REGION Network 47: Ejectors selection
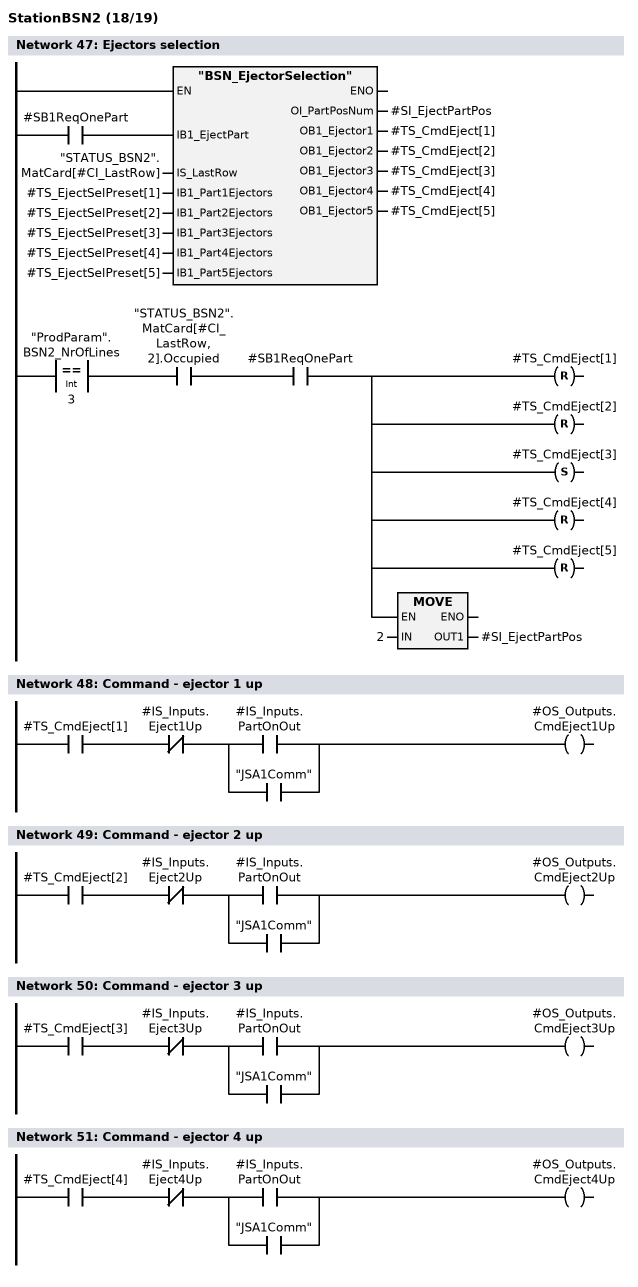
   RUNG wire#powerrail
      "BSN_EjectorSelection"(IB1_EjectPart := wire#w1, IS_LastRow := "STATUS_BSN2".MatCard[#CI_LastRow], IB1_Part1Ejectors := #TS_EjectSelPreset[1], IB1_Part2Ejectors := #TS_EjectSelPreset[2], IB1_Part3Ejectors := #TS_EjectSelPreset[3], IB1_Part4Ejectors := #TS_EjectSelPreset[4], IB1_Part5Ejectors := #TS_EjectSelPreset[5], OI_PartPosNum => #SI_EjectPartPos, OB1_Ejector1 => #TS_CmdEject[1], OB1_Ejector2 => #TS_CmdEject[2], OB1_Ejector3 => #TS_CmdEject[3], OB1_Ejector4 => #TS_CmdEject[4], OB1_Ejector5 => #TS_CmdEject[5])
   END_RUNG
   RUNG wire#powerrail
      Contact( #SB1ReqOnePart )
   END_RUNG wire#w1
   RUNG wire#powerrail
      { S7_Templates := "SrcType := Int" } EQ_Contact(in1 := "ProdParam".BSN2_NrOfLines, in2 := 3)
      Contact( "STATUS_BSN2".MatCard[#CI_LastRow, 2].Occupied )
      Contact( #SB1ReqOnePart )
      wire#w2
      R_Coil( #TS_CmdEject[1] )
   END_RUNG
   RUNG wire#w2
      R_Coil( #TS_CmdEject[2] )
   END_RUNG
   RUNG wire#w2
      S_Coil( #TS_CmdEject[3] )
   END_RUNG
   RUNG wire#w2
      R_Coil( #TS_CmdEject[4] )
   END_RUNG
   RUNG wire#w2
      R_Coil( #TS_CmdEject[5] )
   END_RUNG
   RUNG wire#w2
      Move(in := 2, out1 => #SI_EjectPartPos)
   END_RUNG
   // the same network as SCL:
   "BSN_EjectorSelection"(IB1_EjectPart := #SB1ReqOnePart,
                          IS_LastRow := "STATUS_BSN2".MatCard[#CI_LastRow],
                          IB1_Part1Ejectors := #TS_EjectSelPreset[1],
                          IB1_Part2Ejectors := #TS_EjectSelPreset[2],
                          IB1_Part3Ejectors := #TS_EjectSelPreset[3],
                          IB1_Part4Ejectors := #TS_EjectSelPreset[4],
                          IB1_Part5Ejectors := #TS_EjectSelPreset[5],
                          OI_PartPosNum => #SI_EjectPartPos,
                          OB1_Ejector1 => #TS_CmdEject[1],
                          OB1_Ejector2 => #TS_CmdEject[2],
                          OB1_Ejector3 => #TS_CmdEject[3],
                          OB1_Ejector4 => #TS_CmdEject[4],
                          OB1_Ejector5 => #TS_CmdEject[5]);
   IF ("ProdParam".BSN2_NrOfLines = 3) AND "STATUS_BSN2".MatCard[#CI_LastRow, 2].Occupied AND #SB1ReqOnePart THEN
       #TS_CmdEject[1] := FALSE;
       #TS_CmdEject[2] := FALSE;
       #TS_CmdEject[3] := TRUE;
       #TS_CmdEject[4] := FALSE;
       #TS_CmdEject[5] := FALSE;
       #SI_EjectPartPos := 2;
   END_IF;
END_REGION

REGION Network 48: Command - ejector 1 up
   RUNG wire#powerrail
      Contact( #TS_CmdEject[1] )
      I_Contact( #IS_Inputs.Eject1Up )
      wire#w1
      Contact( #IS_Inputs.PartOnOut )
      wire#w2
      Coil( #OS_Outputs.CmdEject1Up )
   END_RUNG
   RUNG wire#w1
      Contact( "JSA1Comm" )
   END_RUNG wire#w2
   // the same network as SCL:
   #OS_Outputs.CmdEject1Up := #TS_CmdEject[1] AND NOT #IS_Inputs.Eject1Up AND (#IS_Inputs.PartOnOut OR "JSA1Comm");
END_REGION

REGION Network 49: Command - ejector 2 up
   RUNG wire#powerrail
      Contact( #TS_CmdEject[2] )
      I_Contact( #IS_Inputs.Eject2Up )
      wire#w1
      Contact( #IS_Inputs.PartOnOut )
      wire#w2
      Coil( #OS_Outputs.CmdEject2Up )
   END_RUNG
   RUNG wire#w1
      Contact( "JSA1Comm" )
   END_RUNG wire#w2
   // the same network as SCL:
   #OS_Outputs.CmdEject2Up := #TS_CmdEject[2] AND NOT #IS_Inputs.Eject2Up AND (#IS_Inputs.PartOnOut OR "JSA1Comm");
END_REGION

REGION Network 50: Command - ejector 3 up
   RUNG wire#powerrail
      Contact( #TS_CmdEject[3] )
      I_Contact( #IS_Inputs.Eject3Up )
      wire#w1
      Contact( #IS_Inputs.PartOnOut )
      wire#w2
      Coil( #OS_Outputs.CmdEject3Up )
   END_RUNG
   RUNG wire#w1
      Contact( "JSA1Comm" )
   END_RUNG wire#w2
   // the same network as SCL:
   #OS_Outputs.CmdEject3Up := #TS_CmdEject[3] AND NOT #IS_Inputs.Eject3Up AND (#IS_Inputs.PartOnOut OR "JSA1Comm");
END_REGION

REGION Network 51: Command - ejector 4 up
   RUNG wire#powerrail
      Contact( #TS_CmdEject[4] )
      I_Contact( #IS_Inputs.Eject4Up )
      wire#w1
      Contact( #IS_Inputs.PartOnOut )
      wire#w2
      Coil( #OS_Outputs.CmdEject4Up )
   END_RUNG
   RUNG wire#w1
      Contact( "JSA1Comm" )
   END_RUNG wire#w2
   // the same network as SCL:
   #OS_Outputs.CmdEject4Up := #TS_CmdEject[4] AND NOT #IS_Inputs.Eject4Up AND (#IS_Inputs.PartOnOut OR "JSA1Comm");
END_REGION

REGION Network 52: Command - ejector 5 up
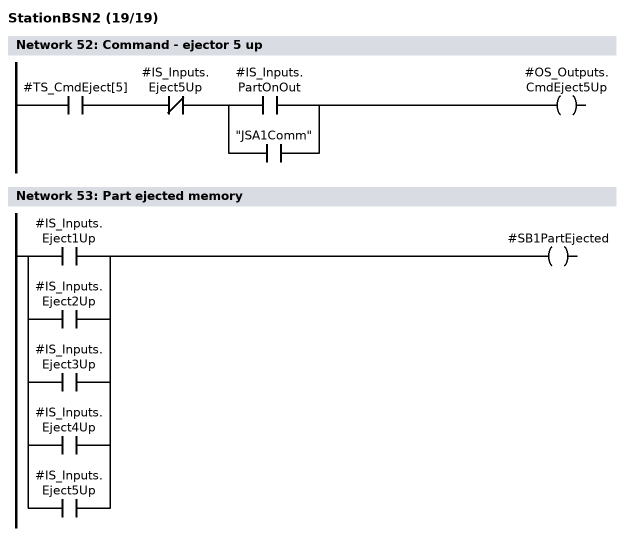
   RUNG wire#powerrail
      Contact( #TS_CmdEject[5] )
      I_Contact( #IS_Inputs.Eject5Up )
      wire#w1
      Contact( #IS_Inputs.PartOnOut )
      wire#w2
      Coil( #OS_Outputs.CmdEject5Up )
   END_RUNG
   RUNG wire#w1
      Contact( "JSA1Comm" )
   END_RUNG wire#w2
   // the same network as SCL:
   #OS_Outputs.CmdEject5Up := #TS_CmdEject[5] AND NOT #IS_Inputs.Eject5Up AND (#IS_Inputs.PartOnOut OR "JSA1Comm");
END_REGION

REGION Network 53: Part ejected memory
   RUNG wire#powerrail
      Contact( #IS_Inputs.Eject1Up )
      wire#w1
      Coil( #SB1PartEjected )
   END_RUNG
   RUNG wire#powerrail
      Contact( #IS_Inputs.Eject2Up )
   END_RUNG wire#w1
   RUNG wire#powerrail
      Contact( #IS_Inputs.Eject3Up )
   END_RUNG wire#w1
   RUNG wire#powerrail
      Contact( #IS_Inputs.Eject4Up )
   END_RUNG wire#w1
   RUNG wire#powerrail
      Contact( #IS_Inputs.Eject5Up )
   END_RUNG wire#w1
   // the same network as SCL:
   #SB1PartEjected := #IS_Inputs.Eject1Up OR #IS_Inputs.Eject2Up OR #IS_Inputs.Eject3Up OR #IS_Inputs.Eject4Up OR #IS_Inputs.Eject5Up;
END_REGION
END_FUNCTION_BLOCK
